(* IEC 61131-3 sources: repolevel_ST_code_completion/output/0127完整版本_带planner/repoeval_Proxy_Application/readful_result_no_provide, 2 files *)

(* ---- Realsubject.st ---- *)
{attribute 'enable_dynamic_creation'}
FUNCTION_BLOCK Realsubject
VAR_INPUT
END_VAR
VAR_OUTPUT
END_VAR
VAR
iProp: INT; // Internal dynamic property for storing the value
END_VAR

METHOD Set_Method : BOOL;
METHOD Get_Method : INT;

END_FUNCTION_BLOCK

// Implementation of the Set_Method
METHOD Set_Method
THIS^.iProp := num;
Set_Method := TRUE;

// Implementation of the Get_Method
METHOD Get_Method
Get_Method := THIS^.iProp;

(* ---- Proxy.st ---- *)
VAR
  // Pointer to store the reference to the subject being protected
  refToRealSubject : POINTER TO Realsubject;
  // Last value of password entered by the client in the visualization element
  iTempPassword : INT;
  // Variable to store the result of the last access attempt
  bLastAccessSuccess : BOOL;
END_VAR
VAR_STAT
  // Default password value for the request to be accepted
  iRealPassword : INT := 1234;
END_VAR

// METHOD fb_init implementation
METHOD fb_init
VAR_INPUT
  bInitRetains : BOOL;
  bInCopyCode : BOOL;
  ptrToRealSubject : POINTER TO Realsubject;
END_VAR
refToRealSubject := ptrToRealSubject;

// METHOD Get_Method implementation
METHOD Get_Method : INT
IF iTempPassword = iRealPassword THEN
  bLastAccessSuccess := TRUE;
  IF refToRealSubject <> 0 THEN
    RETURN refToRealSubject^.iProp;
  END_IF
ELSE
  bLastAccessSuccess := FALSE;
  RETURN -1; // Error code for unauthorized access
END_IF

// METHOD Set_Method implementation
METHOD Set_Method
VAR_INPUT
  num : INT;
END_VAR
IF iTempPassword = iRealPassword THEN
  bLastAccessSuccess := TRUE;
  IF refToRealSubject <> 0 THEN
    refToRealSubject^.iProp := num;
  END_IF
ELSE
  bLastAccessSuccess := FALSE;
END_IF

// METHOD UpdatePassword implementation
METHOD UpdatePassword
VAR_INPUT
  newPassword : INT;
END_VAR
iRealPassword := newPassword;
